// TIA Portal project "automacao_industrial_pick_and_place" (V17)
// Vorlageprojekt für das Buch mit Zielsystem S7-1200

(* hardware
DEVICE "S7-1200-Station_1"  S7-1200 Station
   slot 0: "Baugruppenträger_0"  Rack  V1.0
   slot 1: "PLC_1"  CPU 1217C DC/DC/DC  6ES7 217-1AG40-0XB0  V4.5
*)

// ===== PLC "PLC_1"  CPU 1217C DC/DC/DC =====

VAR_GLOBAL   // PLC tag table "Standard-Variablentabelle"
   "Entry conveyor" AT %A0.0 : Bool;
   "Item at entry" AT %E0.0 : Bool;
   "Item at exit" AT %E0.1 : Bool;
   "Moving X" AT %I0.2 : Bool;
   "Moving Z" AT %I0.3 : Bool;
   "Item detected" AT %I0.4 : Bool;
   "Start" AT %I0.5 : Bool;
   "Reset" AT %I0.6 : Bool;
   "Stop" AT %I0.7 : Bool;
   "Emergency stop" AT %I1.0 : Bool;
   "Auto" AT %I1.1 : Bool;
   "FACTORY I/O (Running)" AT %I1.2 : Bool;
   "Exit conveyor" AT %Q0.1 : Bool;
   "Move X" AT %Q0.2 : Bool;
   "Move Z" AT %Q0.3 : Bool;
   "Grab" AT %Q0.4 : Bool;
   "Start light" AT %Q0.5 : Bool;
   "Reset light" AT %Q0.6 : Bool;
   "Stop light" AT %Q0.7 : Bool;
   "Counter" AT %QW30 : Int;
   "ProcessRunning" AT %M0.0 : Bool;
   "Estado" AT %MW2 : Int;   // Estado atual da maquina
END_VAR

// folder: System blocks/Program resources

DATA_BLOCK "T1"   // DB1
{ S7_Optimized_Access := 'TRUE' }
AUTHOR : Simatic
FAMILY : IEC
NAME : IEC_TMR
VERSION : 1.0
// stored: InstanceOfName IEC_TIMER
"IEC_TIMER"
BEGIN
END_DATA_BLOCK

DATA_BLOCK "T2"   // DB2
{ S7_Optimized_Access := 'TRUE' }
AUTHOR : Simatic
FAMILY : IEC
NAME : IEC_TMR
VERSION : 1.0
// stored: InstanceOfName IEC_TIMER
"IEC_TIMER"
BEGIN
END_DATA_BLOCK

DATA_BLOCK "T3"   // DB3
{ S7_Optimized_Access := 'TRUE' }
AUTHOR : Simatic
FAMILY : IEC
NAME : IEC_TMR
VERSION : 1.0
// stored: InstanceOfName IEC_TIMER
"IEC_TIMER"
BEGIN
END_DATA_BLOCK

// folder: (top level)

FUNCTION "PickAndPlace Logic" : Void   // FC1, LAD
{ S7_Optimized_Access := 'TRUE' }
VERSION : 0.1
BEGIN

REGION Network 1: Liga Sistema
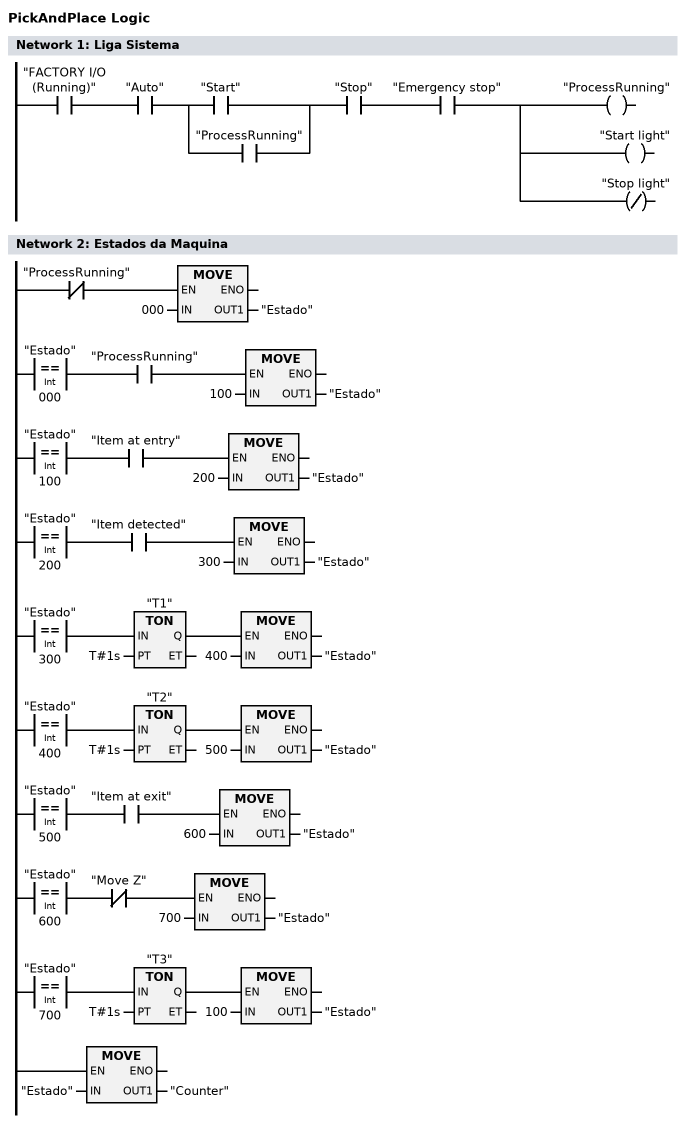
   RUNG wire#powerrail
      Contact( "FACTORY I/O (Running)" )
      Contact( "Auto" )
      wire#w1
      Contact( "Start" )
      wire#w2
      Contact( "Stop" )
      Contact( "Emergency stop" )
      wire#w3
      Coil( "ProcessRunning" )
   END_RUNG
   RUNG wire#w1
      Contact( "ProcessRunning" )
   END_RUNG wire#w2
   RUNG wire#w3
      Coil( "Start light" )
   END_RUNG
   RUNG wire#w3
      I_Coil( "Stop light" )
   END_RUNG
   // the same network as SCL:
   "ProcessRunning" := "FACTORY I/O (Running)" AND "Auto" AND ("Start" OR "ProcessRunning") AND "Stop" AND "Emergency stop";
   "Start light" := "ProcessRunning";
   "Stop light" := NOT "ProcessRunning";
END_REGION

REGION Network 2: Estados da Maquina
   IF NOT "ProcessRunning" THEN "Estado" := 000; END_IF;
   IF ("Estado" = 000) AND "ProcessRunning" THEN "Estado" := 100; END_IF;
   IF ("Estado" = 100) AND "Item at entry" THEN "Estado" := 200; END_IF;
   IF ("Estado" = 200) AND "Item detected" THEN "Estado" := 300; END_IF;
   "T1".TON(IN := "Estado" = 300, PT := T#1s);
   IF "T1".Q THEN "Estado" := 400; END_IF;
   "T2".TON(IN := "Estado" = 400, PT := T#1s);
   IF "T2".Q THEN "Estado" := 500; END_IF;
   IF ("Estado" = 500) AND "Item at exit" THEN "Estado" := 600; END_IF;
   IF ("Estado" = 600) AND NOT "Move Z" THEN "Estado" := 700; END_IF;
   "T3".TON(IN := "Estado" = 700, PT := T#1s);
   IF "T3".Q THEN "Estado" := 100; END_IF;
   "Counter" := "Estado";
END_REGION
END_FUNCTION

ORGANIZATION_BLOCK "Main"   // OB1, FBD, ProgramCycle
TITLE = "Main Program Sweep (Cycle)"
{ S7_Optimized_Access := 'TRUE' }
VERSION : 0.1
   VAR_INPUT
      Initial_Call : Bool;   // Initial call of this OB
      Remanence : Bool;   // =True, if remanent data are available
   END_VAR
BEGIN

REGION Network 1: Konnektierungsbaustein für PLC-Lab
   // Im Netzwerk 1 wird der Konnektierungsbaustein für PLC-Lab aufgerufen.
   // Dieser Aufruf darf nicht entfernt werden!
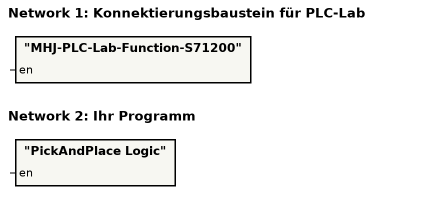
   "MHJ-PLC-Lab-Function-S71200"();
END_REGION

REGION Network 2: Ihr Programm
   // Schreiben Sie ab Netzwerk 2 Ihr Programm
   "PickAndPlace Logic"();
END_REGION
END_ORGANIZATION_BLOCK

// folder: Com

FUNCTION "MHJ-PLC-Lab-Function-S71200" : Void   // FC9000, SCL
{ S7_Optimized_Access := 'TRUE' }
VERSION : 0.1
   VAR_TEMP
      rdTimeReturn : Int;
      outputTime : DTL;
      SyncVal : Byte;
      forVal : Int;
      forVal_2 : Int;
      Value : Byte;
   END_VAR
   VAR CONSTANT
      CompVal : Byte := 16#34;
      Value_01 : Byte := 16#11;
      Value_01_DW : DWord := 16#A165_D992;
      Value_02_DW : DWord := 16#58BE_4401;
   END_VAR
BEGIN

   #Value:=PEEK(area := 16#82,
        dbNumber := 0,
        byteOffset := 511);
   #Value := #Value + 1;

   POKE(area := 16#82,
        dbNumber := 0,
        byteOffset := 511,
        value := #Value);

   POKE(area:=16#81,
        dbNumber:=0,
        byteOffset:=1016,
        value:=#Value_01_DW);
   POKE(area := 16#81,
        dbNumber := 0,
        byteOffset := 1020,
        value := #Value_02_DW);

   POKE(area := 16#81,
        dbNumber := 0,
        byteOffset := 511,
        value := B#16#00);

   FOR #forVal := 0 TO 120 DO
       FOR #forVal_2:=0 TO 10 DO
           #rdTimeReturn:=RD_SYS_T(#outputTime);
           #rdTimeReturn := WR_SYS_T(#outputTime);
           #rdTimeReturn := RD_SYS_T(#outputTime);
           #rdTimeReturn := WR_SYS_T(#outputTime);
       END_FOR;
       #SyncVal:= PEEK(area := 16#81,
                      dbNumber := 0,
                      byteOffset := 511);
       IF #SyncVal = #CompVal THEN
          GOTO M_1;
       END_IF;
   END_FOR;
   RETURN;

   M_1:
   POKE(area := 16#81,
        dbNumber := 0,
        byteOffset := 511,
        value := B#16#0);
END_FUNCTION